// TIA Portal V16 export
// export: Created 2021-11-12T13:31:15.5569335Z, ExportSetting WithDefaults, DisplayName Totally Integrated Automation Portal, DisplayVersion V16 Update 3, DisplayName TIA Portal Version Control Interface, DisplayVersion V16 Update 2, DisplayName TIA Portal Openness, DisplayVersion V16 Update 3, DisplayName SINAMICS Startdrive Advanced, DisplayVersion V16 Update 5, DisplayName SINAMICS Startdrive G130, G150, S120, S150, SINAMICS MV, S210, DisplayVersion V16 Update 5, DisplayName SINAMICS Startdrive G110M, G120, G120C, G120D, G120P, G115D, DisplayVersion V16 Update 5, DisplayName STEP 7 Professional, DisplayVersion V16 Update 3, DisplayName STEP 7 Safety, DisplayVersion V16, DisplayName WinCC UA Professional, DisplayVersion V16 Update 3
FUNCTION "STD_Positioning" : Void   // FC1186, LAD
TITLE = STD_Positioning
{ S7_Optimized_Access := 'TRUE' }
VERSION : 0.1
// Positioning function
// stored: AutoNumber true, IsIECCheckEnabled false, SetENOAutomatically false, UDAEnableTagReadback false
   VAR_INPUT
      IB1PosEn : Bool;   // Positioning mode enable
      IB1Ref : Bool;   // Drive is referenced
      IR_PosValSP : Real;   // Required position (setpoint value)
      IR_PosValAct : Real;   // Actual position
      IR_RoughAppWinSize : Real;   // Window width for rough approaching
      IR_InPosAppWinSize : Real;   // Window width for fine (InPos) approaching
   END_VAR
   VAR_OUTPUT
      OS_Status : "UDT_Positioning_Status";   // Output status
      OB1OutDir1 : Bool;   // Request to run in direction 1 (forward or up)
      OB1OutDir2 : Bool;   // Request to run in direction 2 (reverse or down)
      OB1InRoughApp : Bool;   // Deviation (required pos. - actual pos.) is within the IR_InRoughAppWinSize
      OB1InPosApp : Bool;   // Deviation (required pos. - actual pos.) is within the IR_InPosWinSize
   END_VAR
   VAR_TEMP
      TS_Status : "UDT_Positioning_Status";
      TB1OutDir1 : Bool;   // Request to run in direction 1 (forward or up)
      TB1OutDir2 : Bool;   // Request to run in direction 2 (reverse or down)
      TB1InRoughApp : Bool;   // Deviation (required pos. - actual pos.) is within the IR_InRoughAppWinSize
      TB1InPosApp : Bool;   // Deviation (required pos. - actual pos.) is within the IR_InPosWinSize
      TR_RoughAppPos : Real;
      TR_RoughAppNeg : Real;
      TR_InPosAppPos : Real;
      TR_InPosAppNeg : Real;
      TR_Diff : Real;
   END_VAR
BEGIN

REGION Network 1: Clear temporary variables
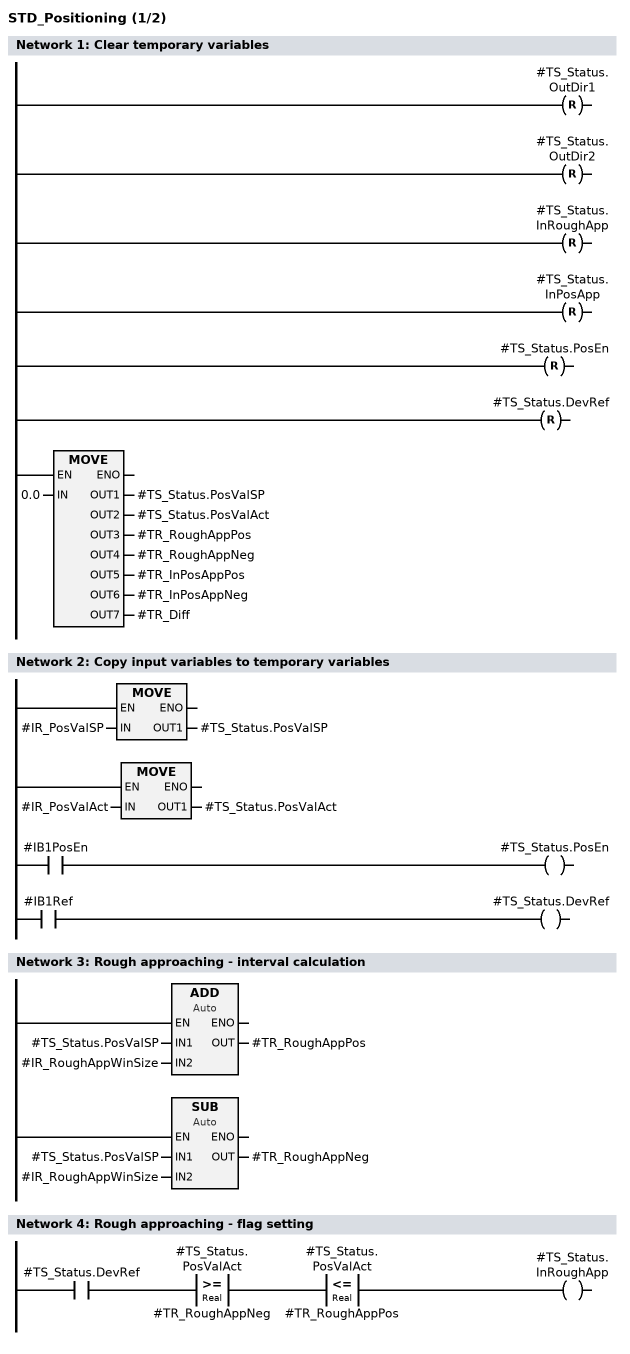
   RUNG wire#powerrail
      R_Coil( #TS_Status.OutDir1 )
   END_RUNG
   RUNG wire#powerrail
      R_Coil( #TS_Status.OutDir2 )
   END_RUNG
   RUNG wire#powerrail
      R_Coil( #TS_Status.InRoughApp )
   END_RUNG
   RUNG wire#powerrail
      R_Coil( #TS_Status.InPosApp )
   END_RUNG
   RUNG wire#powerrail
      R_Coil( #TS_Status.PosEn )
   END_RUNG
   RUNG wire#powerrail
      R_Coil( #TS_Status.DevRef )
   END_RUNG
   RUNG wire#powerrail
      { S7_GenerateENO := "TRUE" } Move(in := 0.0, out1 => #TS_Status.PosValSP, out2 => #TS_Status.PosValAct, out3 => #TR_RoughAppPos, out4 => #TR_RoughAppNeg, out5 => #TR_InPosAppPos, out6 => #TR_InPosAppNeg, out7 => #TR_Diff)
   END_RUNG
   // the same network as SCL:
   #TS_Status.OutDir1 := FALSE;
   #TS_Status.OutDir2 := FALSE;
   #TS_Status.InRoughApp := FALSE;
   #TS_Status.InPosApp := FALSE;
   #TS_Status.PosEn := FALSE;
   #TS_Status.DevRef := FALSE;
   #TS_Status.PosValSP := 0.0;
   #TS_Status.PosValAct := 0.0;
   #TR_RoughAppPos := 0.0;
   #TR_RoughAppNeg := 0.0;
   #TR_InPosAppPos := 0.0;
   #TR_InPosAppNeg := 0.0;
   #TR_Diff := 0.0;
END_REGION

REGION Network 2: Copy input variables to temporary variables
   RUNG wire#powerrail
      { S7_GenerateENO := "TRUE" } Move(in := #IR_PosValSP, out1 => #TS_Status.PosValSP)
   END_RUNG
   RUNG wire#powerrail
      { S7_GenerateENO := "TRUE" } Move(in := #IR_PosValAct, out1 => #TS_Status.PosValAct)
   END_RUNG
   RUNG wire#powerrail
      Contact( #IB1PosEn )
      Coil( #TS_Status.PosEn )
   END_RUNG
   RUNG wire#powerrail
      Contact( #IB1Ref )
      Coil( #TS_Status.DevRef )
   END_RUNG
   // the same network as SCL:
   #TS_Status.PosValSP := #IR_PosValSP;
   #TS_Status.PosValAct := #IR_PosValAct;
   #TS_Status.PosEn := #IB1PosEn;
   #TS_Status.DevRef := #IB1Ref;
END_REGION

REGION Network 3: Rough approaching - interval calculation
   RUNG wire#powerrail
      { S7_GenerateENO := "TRUE" } Add(in1 := #TS_Status.PosValSP, in2 := #IR_RoughAppWinSize, out => #TR_RoughAppPos)
   END_RUNG
   RUNG wire#powerrail
      { S7_GenerateENO := "TRUE" } Sub(in1 := #TS_Status.PosValSP, in2 := #IR_RoughAppWinSize, out => #TR_RoughAppNeg)
   END_RUNG
   // the same network as SCL:
   #TR_RoughAppPos := #TS_Status.PosValSP + #IR_RoughAppWinSize;
   #TR_RoughAppNeg := #TS_Status.PosValSP - #IR_RoughAppWinSize;
END_REGION

REGION Network 4: Rough approaching - flag setting
   RUNG wire#powerrail
      Contact( #TS_Status.DevRef )
      { S7_Templates := "SrcType := Real" } GE_Contact(in1 := #TS_Status.PosValAct, in2 := #TR_RoughAppNeg)
      { S7_Templates := "SrcType := Real" } LE_Contact(in1 := #TS_Status.PosValAct, in2 := #TR_RoughAppPos)
      Coil( #TS_Status.InRoughApp )
   END_RUNG
   // the same network as SCL:
   #TS_Status.InRoughApp := #TS_Status.DevRef AND (#TS_Status.PosValAct >= #TR_RoughAppNeg) AND (#TS_Status.PosValAct <= #TR_RoughAppPos);
END_REGION

REGION Network 5: In position approaching
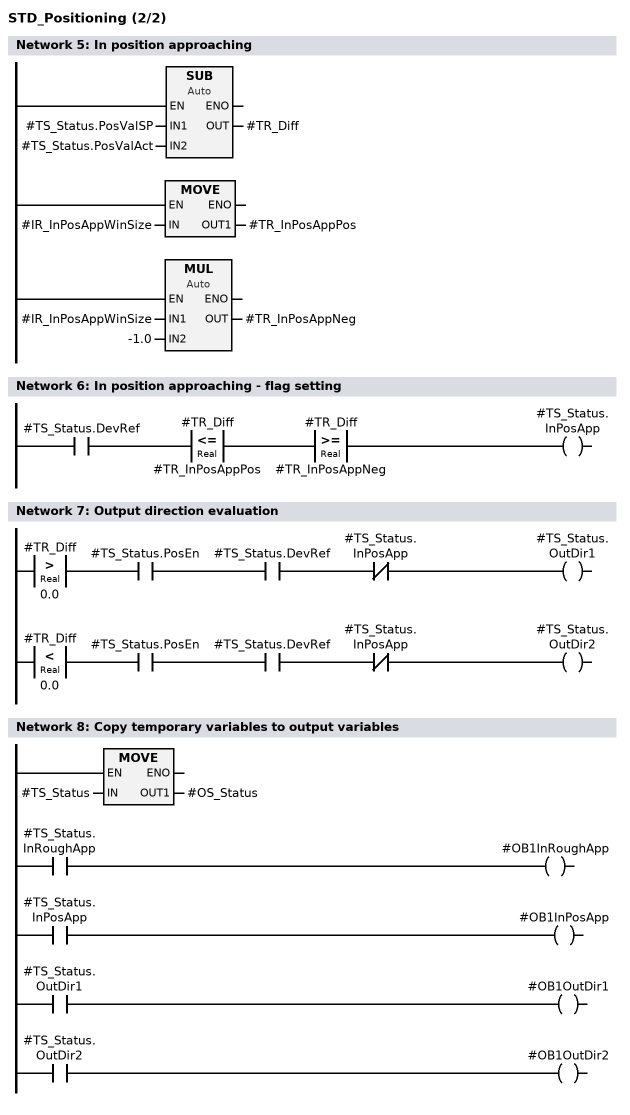
   RUNG wire#powerrail
      { S7_GenerateENO := "TRUE" } Sub(in1 := #TS_Status.PosValSP, in2 := #TS_Status.PosValAct, out => #TR_Diff)
   END_RUNG
   RUNG wire#powerrail
      { S7_GenerateENO := "TRUE" } Move(in := #IR_InPosAppWinSize, out1 => #TR_InPosAppPos)
   END_RUNG
   RUNG wire#powerrail
      { S7_GenerateENO := "TRUE" } Mul(in1 := #IR_InPosAppWinSize, in2 := -1.0, out => #TR_InPosAppNeg)
   END_RUNG
   // the same network as SCL:
   #TR_Diff := #TS_Status.PosValSP - #TS_Status.PosValAct;
   #TR_InPosAppPos := #IR_InPosAppWinSize;
   #TR_InPosAppNeg := #IR_InPosAppWinSize * (-1.0);
END_REGION

REGION Network 6: In position approaching - flag setting
   RUNG wire#powerrail
      Contact( #TS_Status.DevRef )
      { S7_Templates := "SrcType := Real" } LE_Contact(in1 := #TR_Diff, in2 := #TR_InPosAppPos)
      { S7_Templates := "SrcType := Real" } GE_Contact(in1 := #TR_Diff, in2 := #TR_InPosAppNeg)
      Coil( #TS_Status.InPosApp )
   END_RUNG
   // the same network as SCL:
   #TS_Status.InPosApp := #TS_Status.DevRef AND (#TR_Diff <= #TR_InPosAppPos) AND (#TR_Diff >= #TR_InPosAppNeg);
END_REGION

REGION Network 7: Output direction evaluation
   RUNG wire#powerrail
      { S7_Templates := "SrcType := Real" } GT_Contact(in1 := #TR_Diff, in2 := 0.0)
      Contact( #TS_Status.PosEn )
      Contact( #TS_Status.DevRef )
      I_Contact( #TS_Status.InPosApp )
      Coil( #TS_Status.OutDir1 )
   END_RUNG
   RUNG wire#powerrail
      { S7_Templates := "SrcType := Real" } LT_Contact(in1 := #TR_Diff, in2 := 0.0)
      Contact( #TS_Status.PosEn )
      Contact( #TS_Status.DevRef )
      I_Contact( #TS_Status.InPosApp )
      Coil( #TS_Status.OutDir2 )
   END_RUNG
   // the same network as SCL:
   #TS_Status.OutDir1 := (#TR_Diff > 0.0) AND #TS_Status.PosEn AND #TS_Status.DevRef AND NOT #TS_Status.InPosApp;
   #TS_Status.OutDir2 := (#TR_Diff < 0.0) AND #TS_Status.PosEn AND #TS_Status.DevRef AND NOT #TS_Status.InPosApp;
END_REGION

REGION Network 8: Copy temporary variables to output variables
   RUNG wire#powerrail
      { S7_GenerateENO := "TRUE" } Move(in := #TS_Status, out1 => #OS_Status)
   END_RUNG
   RUNG wire#powerrail
      Contact( #TS_Status.InRoughApp )
      Coil( #OB1InRoughApp )
   END_RUNG
   RUNG wire#powerrail
      Contact( #TS_Status.InPosApp )
      Coil( #OB1InPosApp )
   END_RUNG
   RUNG wire#powerrail
      Contact( #TS_Status.OutDir1 )
      Coil( #OB1OutDir1 )
   END_RUNG
   RUNG wire#powerrail
      Contact( #TS_Status.OutDir2 )
      Coil( #OB1OutDir2 )
   END_RUNG
   // the same network as SCL:
   #OS_Status := #TS_Status;
   #OB1InRoughApp := #TS_Status.InRoughApp;
   #OB1InPosApp := #TS_Status.InPosApp;
   #OB1OutDir1 := #TS_Status.OutDir1;
   #OB1OutDir2 := #TS_Status.OutDir2;
END_REGION
END_FUNCTION
